TEXTLIST PML_Modes_txt
  0 = 'Undefined'
  1 = 'Production'
  2 = 'Manual'
   = ''
END_TEXTLIST

(* stored: Version 1.1.0.1, ProductVersion 3.1.4024.11
   TextList PML_Modes_txt: Id {ff34e805-28b9-4e08-814c-85b86aaaf3db} *)
